TYPE E_MatchedSlaveArmIdx :
(
	MatchedSlaveArmIdx_NULL := 0,
	MatchedSlaveArmIdx_1 := 1,
	MatchedSlaveArmIdx_2 := 2,
	MatchedSlaveArmIdx_3 := 3,
	MatchedSlaveArmIdx_4 := 4
);
END_TYPE

(* stored: Version 1.1.0.1, ProductVersion 3.1.4024.12
   DUT E_MatchedSlaveArmIdx: Id {4bff68be-f9ee-4383-8597-63c0b5507430} *)
